FUNCTION_BLOCK MultiNeredaCmd (* Composite Function Block Type *)
  (* Standard: 61499-2 *)
  (* Version 0.0, 6/9/2026, Schneider Electric, template *)
  PACKAGE SE.Nereda;
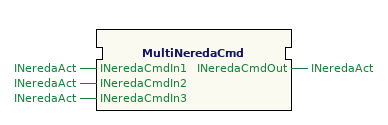
  SOCKETS
    INeredaCmdIn1 : INeredaAct;
    INeredaCmdIn2 : INeredaAct;
    INeredaCmdIn3 : INeredaAct;
  END_SOCKETS
  PLUGS
    INeredaCmdOut : INeredaAct;
  END_PLUGS
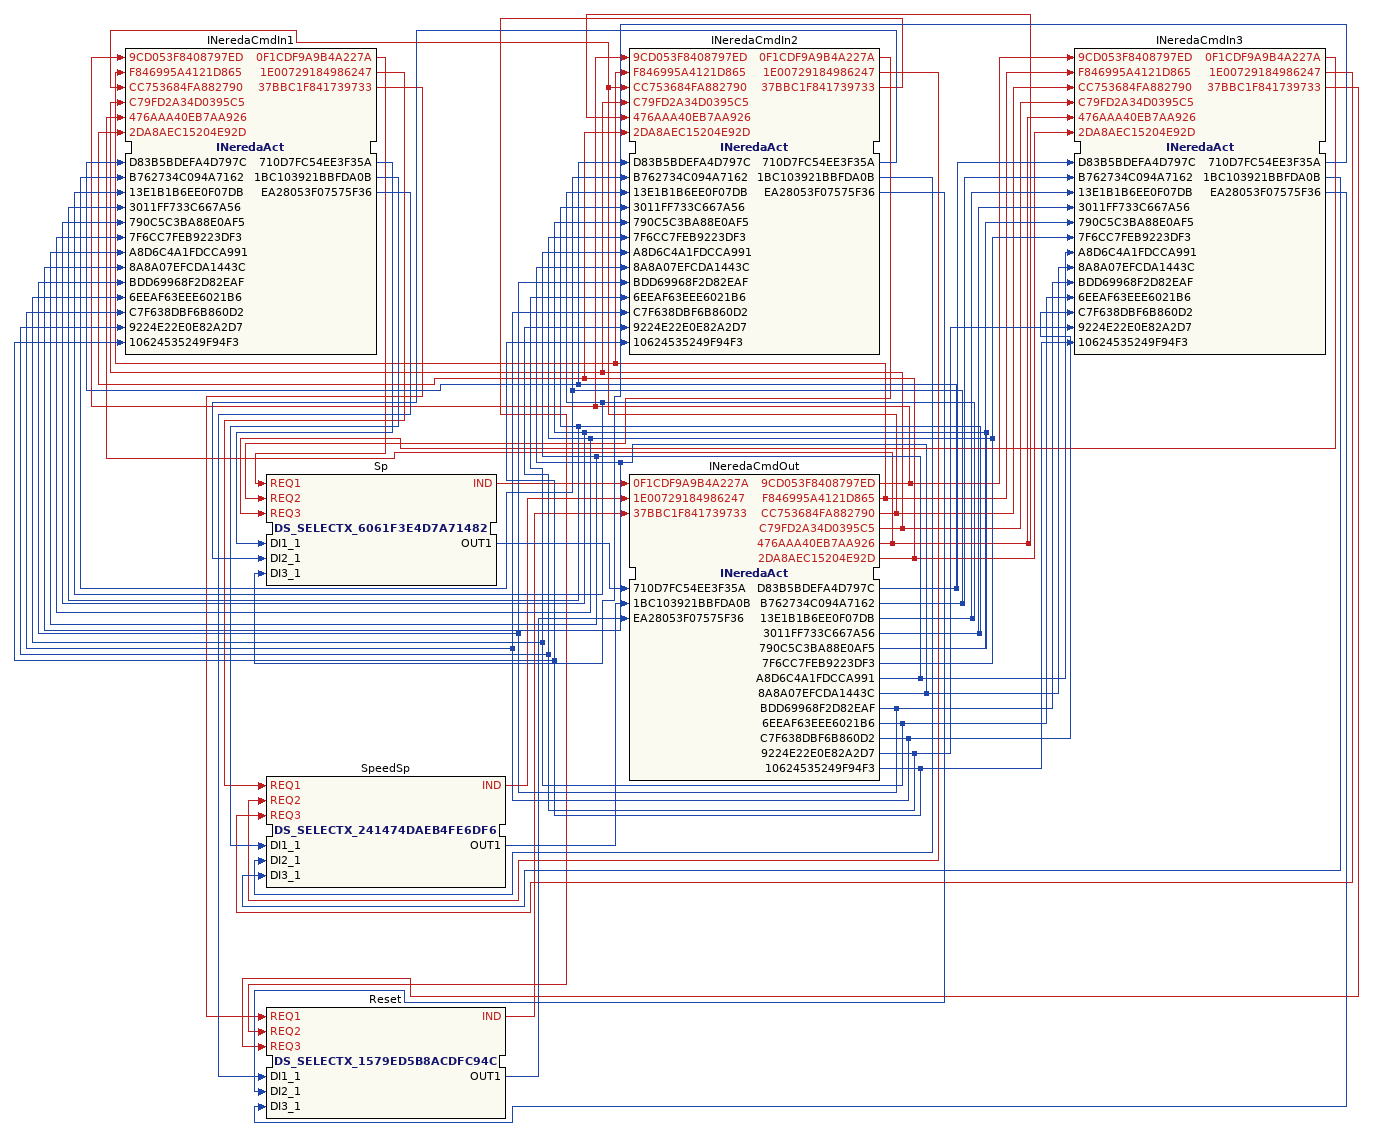
  FBS
    Sp : DS_SELECTX_6061F3E4D7A71482; {SET_ATTRIBUTE(Configuration.GenericFBType.InterfaceParams, Runtime.Standard#CNTX:=3;CNTY:=1;DI${CNTX,_,CNTY$}:INT)}
    SpeedSp : DS_SELECTX_241474DAEB4FE6DF6; {SET_ATTRIBUTE(Configuration.GenericFBType.InterfaceParams, Runtime.Standard#CNTX:=3;CNTY:=1;DI${CNTX,_,CNTY$}:REAL)}
    Reset : DS_SELECTX_1579ED5B8ACDFC94C; {SET_ATTRIBUTE(Configuration.GenericFBType.InterfaceParams, Runtime.Standard#CNTX:=3;CNTY:=1;DI${CNTX,_,CNTY$}:BOOL)}
  END_FBS
  EVENT_CONNECTIONS
    Sp.IND TO INeredaCmdOut.0F1CDF9A9B4A227A;
    SpeedSp.IND TO INeredaCmdOut.1E00729184986247;
    Reset.IND TO INeredaCmdOut.37BBC1F841739733;
    INeredaCmdOut.9CD053F8408797ED TO INeredaCmdIn1.9CD053F8408797ED;
    INeredaCmdOut.F846995A4121D865 TO INeredaCmdIn1.F846995A4121D865;
    INeredaCmdOut.CC753684FA882790 TO INeredaCmdIn1.CC753684FA882790;
    INeredaCmdOut.C79FD2A34D0395C5 TO INeredaCmdIn1.C79FD2A34D0395C5;
    INeredaCmdOut.476AAA40EB7AA926 TO INeredaCmdIn1.476AAA40EB7AA926;
    INeredaCmdOut.2DA8AEC15204E92D TO INeredaCmdIn1.2DA8AEC15204E92D;
    INeredaCmdOut.9CD053F8408797ED TO INeredaCmdIn2.9CD053F8408797ED;
    INeredaCmdOut.F846995A4121D865 TO INeredaCmdIn2.F846995A4121D865;
    INeredaCmdOut.CC753684FA882790 TO INeredaCmdIn2.CC753684FA882790;
    INeredaCmdOut.C79FD2A34D0395C5 TO INeredaCmdIn2.C79FD2A34D0395C5;
    INeredaCmdOut.476AAA40EB7AA926 TO INeredaCmdIn2.476AAA40EB7AA926;
    INeredaCmdOut.2DA8AEC15204E92D TO INeredaCmdIn2.2DA8AEC15204E92D;
    INeredaCmdOut.9CD053F8408797ED TO INeredaCmdIn3.9CD053F8408797ED;
    INeredaCmdOut.F846995A4121D865 TO INeredaCmdIn3.F846995A4121D865;
    INeredaCmdOut.CC753684FA882790 TO INeredaCmdIn3.CC753684FA882790;
    INeredaCmdOut.C79FD2A34D0395C5 TO INeredaCmdIn3.C79FD2A34D0395C5;
    INeredaCmdOut.476AAA40EB7AA926 TO INeredaCmdIn3.476AAA40EB7AA926;
    INeredaCmdOut.2DA8AEC15204E92D TO INeredaCmdIn3.2DA8AEC15204E92D;
    INeredaCmdIn1.0F1CDF9A9B4A227A TO Sp.REQ1;
    INeredaCmdIn1.1E00729184986247 TO SpeedSp.REQ1;
    INeredaCmdIn1.37BBC1F841739733 TO Reset.REQ1;
    INeredaCmdIn2.0F1CDF9A9B4A227A TO Sp.REQ2;
    INeredaCmdIn2.1E00729184986247 TO SpeedSp.REQ2;
    INeredaCmdIn2.37BBC1F841739733 TO Reset.REQ2;
    INeredaCmdIn3.0F1CDF9A9B4A227A TO Sp.REQ3;
    INeredaCmdIn3.1E00729184986247 TO SpeedSp.REQ3;
    INeredaCmdIn3.37BBC1F841739733 TO Reset.REQ3;
  END_CONNECTIONS
  DATA_CONNECTIONS
    Sp.OUT1 TO INeredaCmdOut.710D7FC54EE3F35A;
    SpeedSp.OUT1 TO INeredaCmdOut.1BC103921BBFDA0B;
    Reset.OUT1 TO INeredaCmdOut.EA28053F07575F36;
    INeredaCmdOut.D83B5BDEFA4D797C TO INeredaCmdIn1.D83B5BDEFA4D797C;
    INeredaCmdOut.B762734C094A7162 TO INeredaCmdIn1.B762734C094A7162;
    INeredaCmdOut.13E1B1B6EE0F07DB TO INeredaCmdIn1.13E1B1B6EE0F07DB;
    INeredaCmdOut.3011FF733C667A56 TO INeredaCmdIn1.3011FF733C667A56;
    INeredaCmdOut.790C5C3BA88E0AF5 TO INeredaCmdIn1.790C5C3BA88E0AF5;
    INeredaCmdOut.7F6CC7FEB9223DF3 TO INeredaCmdIn1.7F6CC7FEB9223DF3;
    INeredaCmdOut.A8D6C4A1FDCCA991 TO INeredaCmdIn1.A8D6C4A1FDCCA991;
    INeredaCmdOut.8A8A07EFCDA1443C TO INeredaCmdIn1.8A8A07EFCDA1443C;
    INeredaCmdOut.BDD69968F2D82EAF TO INeredaCmdIn1.BDD69968F2D82EAF;
    INeredaCmdOut.6EEAF63EEE6021B6 TO INeredaCmdIn1.6EEAF63EEE6021B6;
    INeredaCmdOut.C7F638DBF6B860D2 TO INeredaCmdIn1.C7F638DBF6B860D2;
    INeredaCmdOut.9224E22E0E82A2D7 TO INeredaCmdIn1.9224E22E0E82A2D7;
    INeredaCmdOut.10624535249F94F3 TO INeredaCmdIn1.10624535249F94F3;
    INeredaCmdOut.D83B5BDEFA4D797C TO INeredaCmdIn2.D83B5BDEFA4D797C;
    INeredaCmdOut.B762734C094A7162 TO INeredaCmdIn2.B762734C094A7162;
    INeredaCmdOut.13E1B1B6EE0F07DB TO INeredaCmdIn2.13E1B1B6EE0F07DB;
    INeredaCmdOut.3011FF733C667A56 TO INeredaCmdIn2.3011FF733C667A56;
    INeredaCmdOut.790C5C3BA88E0AF5 TO INeredaCmdIn2.790C5C3BA88E0AF5;
    INeredaCmdOut.7F6CC7FEB9223DF3 TO INeredaCmdIn2.7F6CC7FEB9223DF3;
    INeredaCmdOut.A8D6C4A1FDCCA991 TO INeredaCmdIn2.A8D6C4A1FDCCA991;
    INeredaCmdOut.8A8A07EFCDA1443C TO INeredaCmdIn2.8A8A07EFCDA1443C;
    INeredaCmdOut.BDD69968F2D82EAF TO INeredaCmdIn2.BDD69968F2D82EAF;
    INeredaCmdOut.6EEAF63EEE6021B6 TO INeredaCmdIn2.6EEAF63EEE6021B6;
    INeredaCmdOut.C7F638DBF6B860D2 TO INeredaCmdIn2.C7F638DBF6B860D2;
    INeredaCmdOut.9224E22E0E82A2D7 TO INeredaCmdIn2.9224E22E0E82A2D7;
    INeredaCmdOut.10624535249F94F3 TO INeredaCmdIn2.10624535249F94F3;
    INeredaCmdOut.D83B5BDEFA4D797C TO INeredaCmdIn3.D83B5BDEFA4D797C;
    INeredaCmdOut.B762734C094A7162 TO INeredaCmdIn3.B762734C094A7162;
    INeredaCmdOut.13E1B1B6EE0F07DB TO INeredaCmdIn3.13E1B1B6EE0F07DB;
    INeredaCmdOut.3011FF733C667A56 TO INeredaCmdIn3.3011FF733C667A56;
    INeredaCmdOut.790C5C3BA88E0AF5 TO INeredaCmdIn3.790C5C3BA88E0AF5;
    INeredaCmdOut.7F6CC7FEB9223DF3 TO INeredaCmdIn3.7F6CC7FEB9223DF3;
    INeredaCmdOut.A8D6C4A1FDCCA991 TO INeredaCmdIn3.A8D6C4A1FDCCA991;
    INeredaCmdOut.8A8A07EFCDA1443C TO INeredaCmdIn3.8A8A07EFCDA1443C;
    INeredaCmdOut.BDD69968F2D82EAF TO INeredaCmdIn3.BDD69968F2D82EAF;
    INeredaCmdOut.6EEAF63EEE6021B6 TO INeredaCmdIn3.6EEAF63EEE6021B6;
    INeredaCmdOut.C7F638DBF6B860D2 TO INeredaCmdIn3.C7F638DBF6B860D2;
    INeredaCmdOut.9224E22E0E82A2D7 TO INeredaCmdIn3.9224E22E0E82A2D7;
    INeredaCmdOut.10624535249F94F3 TO INeredaCmdIn3.10624535249F94F3;
    INeredaCmdIn1.710D7FC54EE3F35A TO Sp.DI1_1;
    INeredaCmdIn1.1BC103921BBFDA0B TO SpeedSp.DI1_1;
    INeredaCmdIn1.EA28053F07575F36 TO Reset.DI1_1;
    INeredaCmdIn2.710D7FC54EE3F35A TO Sp.DI2_1;
    INeredaCmdIn2.1BC103921BBFDA0B TO SpeedSp.DI2_1;
    INeredaCmdIn2.EA28053F07575F36 TO Reset.DI2_1;
    INeredaCmdIn3.710D7FC54EE3F35A TO Sp.DI3_1;
    INeredaCmdIn3.1BC103921BBFDA0B TO SpeedSp.DI3_1;
    INeredaCmdIn3.EA28053F07575F36 TO Reset.DI3_1;
  END_CONNECTIONS
END_FUNCTION_BLOCK
